Staubli VAL3: deleteFile.pgx

program deleteFile()
  local bool l_bRes
begin
  //delete the file or folder
  l_bRes=$delete(sFileDelete)
  if l_bRes
    gotoxy(1,2)
    put("删除:"+sFileDelete)
  else
    gotoxy(1,2)
    put("删除:失败"+sFileDelete)
  endIf

end
